(* PLC project CoDeSys External Library Template, WAGO e!COCKPIT e!COCKPIT, author 3S - Smart Software Solutions GmbH *)
(* stored: creationDateTime 2019-10-29T12:37:19.9024695, version 3.5.5.30, modificationDateTime 2019-10-29T12:36:39.3744516, organization 3S - Smart Software Solutions GmbH *)
(* Library project template with all possible element types, docu and a sample project structure *)

FUNCTION fnKomunikatSprawdzTimeStamp : STRING
  VAR_INPUT
    sKomunikat : alSTRINGKomunikat;
  END_VAR
  VAR_IN_OUT
    dtDataCzasWKomunikacie : DT;
    dtDataCzasAktualny : DT;
  END_VAR
  VAR
    sKomunikatDoObrobki : alSTRINGKomunikat;
    sString : STRING;
    uintRok : UINT;
    uintMiesiac : UINT;
    uintDzien : UINT;
    uintGodzina : UINT;
    uintMinuta : UINT;
    uintSekunda : UINT;
  END_VAR

            sKomunikatDoObrobki := sKomunikat;

sString := 'DT#'; 
sString := CONCAT(sString, MID(sKomunikatDoObrobki, 10, 48));
sString := CONCAT(sString, '-'); 
sString := CONCAT(sString, MID(sKomunikatDoObrobki, 8, 59)); 
dtDataCzasWKomunikacie := STRING_TO_DT(sString);
dtDataCzasAktualny := FuGetDateAndTime();

fnKomunikatSprawdzTimeStamp := sString;
          
END_FUNCTION
